// Mitsubishi GX Works2 project: ZP_funtion2   PLC: Q03UDV

PROGRAM MAIN
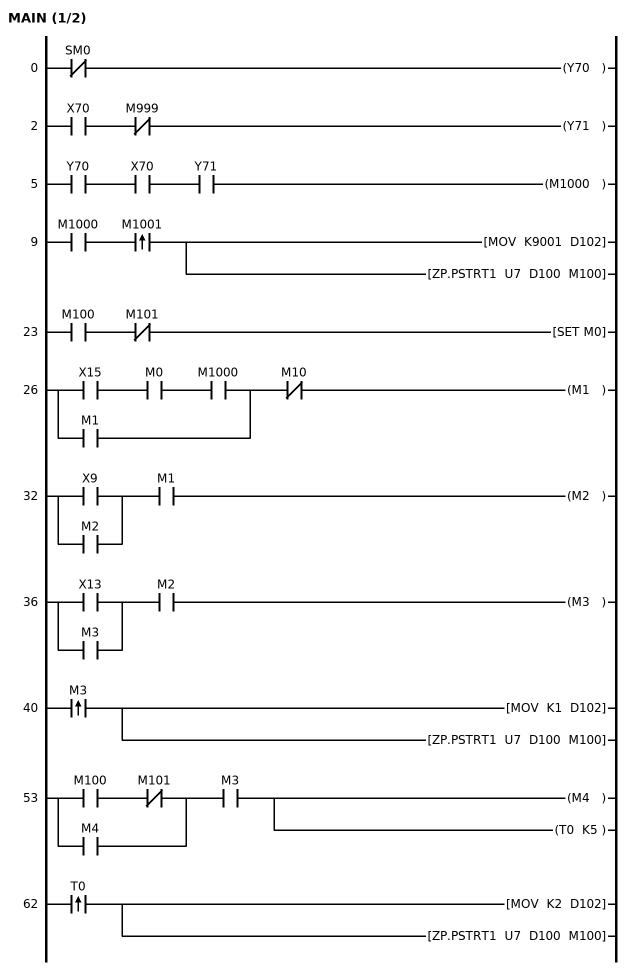
0     LDI     SM0
      OUT     Y70
2     LD      X70
      ANI     M999
      OUT     Y71
5     LD      Y70
      AND     X70
      AND     Y71
      OUT     M1000
9     LD      M1000
      ANDP    M1001
      MOV     K9001 D102
      ZP.PSTRT1 U7 D100 M100
23    LD      M100
      ANI     M101
      SET     M0
26    LD      X15
      AND     M0
      AND     M1000
      OR      M1
      ANI     M10
      OUT     M1
32    LD      X9
      OR      M2
      AND     M1
      OUT     M2
36    LD      X13
      OR      M3
      AND     M2
      OUT     M3
40    LDP     M3
      MOV     K1 D102
      ZP.PSTRT1 U7 D100 M100
53    LD      M100
      ANI     M101
      OR      M4
      AND     M3
      OUT     M4
      OUT     T0 K5
62    LDP     T0
      MOV     K2 D102
      ZP.PSTRT1 U7 D100 M100
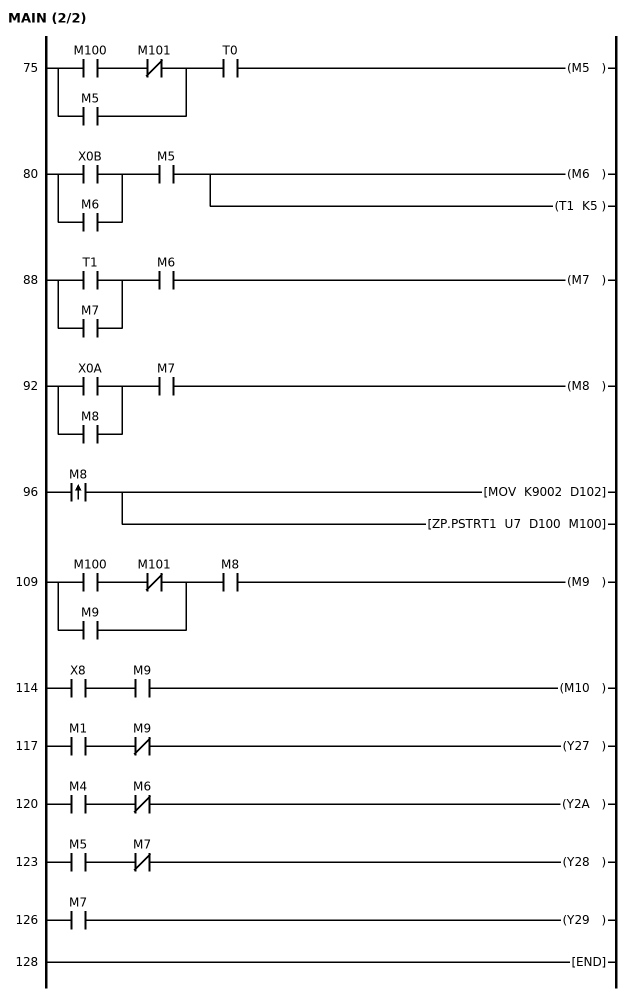
75    LD      M100
      ANI     M101
      OR      M5
      AND     T0
      OUT     M5
80    LD      X0B
      OR      M6
      AND     M5
      OUT     M6
      OUT     T1 K5
88    LD      T1
      OR      M7
      AND     M6
      OUT     M7
92    LD      X0A
      OR      M8
      AND     M7
      OUT     M8
96    LDP     M8
      MOV     K9002 D102
      ZP.PSTRT1 U7 D100 M100
109   LD      M100
      ANI     M101
      OR      M9
      AND     M8
      OUT     M9
114   LD      X8
      AND     M9
      OUT     M10
117   LD      M1
      ANI     M9
      OUT     Y27
120   LD      M4
      ANI     M6
      OUT     Y2A
123   LD      M5
      ANI     M7
      OUT     Y28
126   LD      M7
      OUT     Y29
128   END
END_PROGRAM
